// TIA Portal V18 export
// export: Created 2026-03-12T16:04:34.4113994Z, ExportSetting WithDefaults, DisplayName Totally Integrated Automation Portal, DisplayVersion V18 Update 5, DisplayName TIA Portal Openness, DisplayVersion V18 Update 5, DisplayName TIA Portal Version Control Interface, DisplayVersion V18, DisplayName SINAMICS Startdrive Advanced, DisplayVersion V18, DisplayName SINAMICS Startdrive G130, G150, S120, S150, SINAMICS MV, S210, DisplayVersion V18, DisplayName SINAMICS Startdrive G110M, G120, G120C, G120D, G120P, G115D, DisplayVersion V18, DisplayName STEP 7 Professional, DisplayVersion V18 Update 5, DisplayName STEP 7 Safety, DisplayVersion V18, DisplayName WinCC Professional, DisplayVersion V18 Update 5
FUNCTION_BLOCK "FB MODOS DE OPERAÇÃO"   // FB10, LAD
TITLE = Function Block MODOS DE OPERAÇÃO
{ S7_Optimized_Access := 'TRUE' }
VERSION : 0.1
// Movendo os valores booleados para uma variável do tipo int
// stored: AutoNumber true, IsIECCheckEnabled false, IsRetainMemResEnabled false, MemoryReserve 100, SetENOAutomatically false, UDAEnableTagReadback false
   VAR_INPUT
      INPUT_RM : Bool;   // Entrada de sinal alto para indicar modo Remoto Manual
      INPUT_RA : Bool;   // Entrada de sinal alto para indicar modo Remoto Automático
      INPUT_LM : Bool;   // Entrada de sinal alto para indicar modo Local Manual
      INPUT_LA : Bool;   // Entrada de sinal alto para indicar modo Local Automático
   END_VAR
   VAR_OUTPUT
      OUTPUT_MODO : Int;   // Saída do Modo de Operação
   END_VAR
BEGIN

REGION Network 1: Estrutura de Operação
   // Se Remoto Manual = TRUE, OPERACAO_MOTOR = 1 
   // Se Remoto Automático = TRUE, OPERACAO_MOTOR = 2
   // Se Local Automático = TRUE, OPERACAO_MOTOR = 3
   // Se Local Manual = TRUE, OPERACAO_MOTOR = 4
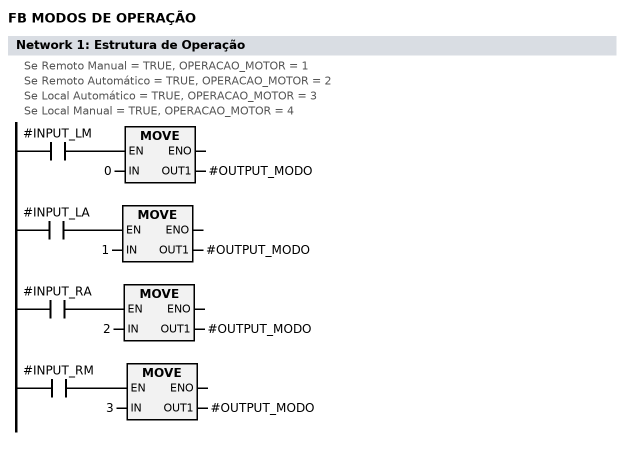
   RUNG wire#powerrail
      Contact( #INPUT_LM )
      Move(in := 0, out1 => #OUTPUT_MODO)
   END_RUNG
   RUNG wire#powerrail
      Contact( #INPUT_LA )
      Move(in := 1, out1 => #OUTPUT_MODO)
   END_RUNG
   RUNG wire#powerrail
      Contact( #INPUT_RA )
      Move(in := 2, out1 => #OUTPUT_MODO)
   END_RUNG
   RUNG wire#powerrail
      Contact( #INPUT_RM )
      Move(in := 3, out1 => #OUTPUT_MODO)
   END_RUNG
   // the same network as SCL:
   IF #INPUT_LM THEN #OUTPUT_MODO := 0; END_IF;
   IF #INPUT_LA THEN #OUTPUT_MODO := 1; END_IF;
   IF #INPUT_RA THEN #OUTPUT_MODO := 2; END_IF;
   IF #INPUT_RM THEN #OUTPUT_MODO := 3; END_IF;
END_REGION
END_FUNCTION_BLOCK
